Yaskawa INFORM job: kufsa_test_250.JBI

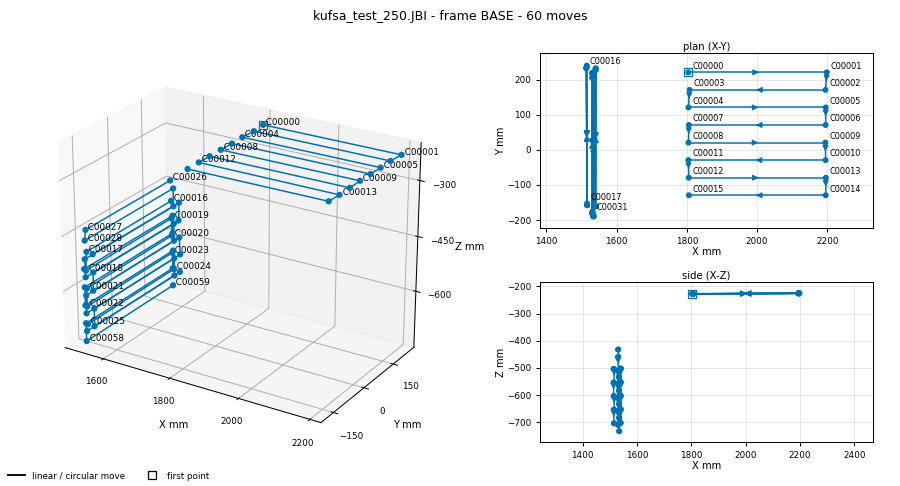
[picture p0: tool path of kufsa_test_250.JBI in frame BASE, 60 of 65 moves have a stored position in this frame; points joined in program order, loops and branches not executed]
/JOB
//NAME kufsa_test_250
//POS
///NPOS 60,0,60,0,0,0
///TOOL 0
///POSTYPE BASE
///RECTAN
///RCONF 0,0,0,0,0,0,0,0,0,0,0,0,0,0,0,0,0,0,0,0,0,0,0,0
C00000=1804.266,220.599,-227.332,179.0000,1.0000,1.0000
C00001=2198.370,220.599,-225.837,179.0000,1.0000,1.0000
C00002=2194.801,170.599,-225.649,179.0000,1.0000,1.0000
C00003=1807.577,170.599,-227.559,179.0000,1.0000,1.0000
C00004=1804.622,120.599,-227.769,179.0000,1.0000,1.0000
C00005=2195.335,120.599,-225.843,179.0000,1.0000,1.0000
C00006=2195.106,70.599,-225.320,179.0000,1.0000,1.0000
C00007=1805.716,70.599,-228.029,179.0000,1.0000,1.0000
C00008=1804.735,20.599,-228.045,179.0000,1.0000,1.0000
C00009=2194.418,20.599,-225.391,179.0000,1.0000,1.0000
C00010=2195.097,-29.400,-225.681,179.0000,1.0000,1.0000
C00011=1804.440,-29.400,-228.141,179.0000,1.0000,1.0000
C00012=1805.619,-79.400,-227.256,179.0000,1.0000,1.0000
C00013=2195.630,-79.400,-225.700,179.0000,1.0000,1.0000
C00014=2195.292,-129.400,-224.241,179.0000,1.0000,1.0000
C00015=1805.953,-129.400,-227.208,179.0000,1.0000,1.0000
C00016=1513.631,232.354,-503.993,179.0000,-89.9999,1.0000
C00017=1516.149,-153.231,-503.993,179.0000,-89.9999,1.0000
C00018=1516.042,-157.471,-553.993,179.0000,-89.9999,1.0000
C00019=1513.923,233.133,-553.993,179.0000,-89.9999,1.0000
C00020=1514.033,233.523,-603.993,179.0000,-89.9999,1.0000
C00021=1516.196,-156.884,-603.993,179.0000,-89.9999,1.0000
C00022=1516.145,-156.999,-653.993,179.0000,-89.9999,1.0000
C00023=1514.649,233.710,-653.993,179.0000,-89.9999,1.0000
C00024=1515.282,239.938,-703.993,179.0000,-89.9999,1.0000
C00025=1516.324,-157.007,-703.993,179.0000,-89.9999,1.0000
C00026=1530.443,204.779,-432.522,179.0000,-89.9999,1.0000
C00027=1531.499,-175.214,-432.522,179.0000,-89.9999,1.0000
C00028=1531.405,-179.918,-459.727,179.0000,-89.9999,1.0000
C00029=1530.485,218.119,-459.727,179.0000,-89.9999,1.0000
C00030=1531.882,216.269,-509.727,179.0000,-89.9999,1.0000
C00031=1531.275,-181.949,-509.727,179.0000,-89.9999,1.0000
C00032=1531.305,-180.389,-559.727,179.0000,-89.9999,1.0000
C00033=1531.688,217.320,-559.727,179.0000,-89.9999,1.0000
C00034=1530.439,218.736,-609.727,179.0000,-89.9999,1.0000
C00035=1531.606,-180.718,-609.727,179.0000,-89.9999,1.0000
C00036=1530.852,-180.562,-659.727,179.0000,-89.9999,1.0000
C00037=1531.645,217.737,-659.727,179.0000,-89.9999,1.0000
C00038=1532.334,216.222,-709.727,179.0000,-89.9999,1.0000
C00039=1530.209,-180.083,-709.727,179.0000,-89.9999,1.0000
C00040=1540.494,-160.372,-502.282,179.0000,-89.9999,1.0000
C00041=1540.352,230.020,-502.282,179.0000,-89.9999,1.0000
C00042=1540.533,226.582,-552.282,179.0000,-89.9999,1.0000
C00043=1540.232,-160.082,-552.282,179.0000,-89.9999,1.0000
C00044=1539.904,-161.733,-602.282,179.0000,-89.9999,1.0000
C00045=1540.218,229.622,-602.282,179.0000,-89.9999,1.0000
C00046=1540.573,232.252,-652.282,179.0000,-89.9999,1.0000
C00047=1540.340,-160.160,-652.282,179.0000,-89.9999,1.0000
C00048=1539.291,-159.918,-702.282,179.0000,-89.9999,1.0000
C00049=1540.509,230.302,-702.282,179.0000,-89.9999,1.0000
C00050=1534.042,-189.208,-533.001,179.0000,-89.9999,1.0000
C00051=1534.110,208.321,-533.001,179.0000,-89.9999,1.0000
C00052=1533.962,207.490,-583.001,179.0000,-89.9999,1.0000
C00053=1534.342,-189.439,-583.001,179.0000,-89.9999,1.0000
C00054=1534.609,-189.394,-633.001,179.0000,-89.9999,1.0000
C00055=1534.722,207.440,-633.001,179.0000,-89.9999,1.0000
C00056=1535.013,204.575,-683.001,179.0000,-89.9999,1.0000
C00057=1534.488,-188.796,-683.001,179.0000,-89.9999,1.0000
C00058=1534.671,-189.015,-733.001,179.0000,-89.9999,1.0000
C00059=1535.183,204.586,-733.001,179.0000,-89.9999,1.0000
///POSTYPE PULSE
///PULSE
EC00000=0
EC00001=0
EC00002=0
EC00003=0
EC00004=0
EC00005=0
EC00006=0
EC00007=0
EC00008=0
EC00009=0
EC00010=0
EC00011=0
EC00012=0
EC00013=0
EC00014=0
EC00015=0
EC00016=0
EC00017=0
EC00018=0
EC00019=0
EC00020=0
EC00021=0
EC00022=0
EC00023=0
EC00024=0
EC00025=0
EC00026=92160
EC00027=92160
EC00028=92160
EC00029=92160
EC00030=92160
EC00031=92160
EC00032=92160
EC00033=92160
EC00034=92160
EC00035=92160
EC00036=92160
EC00037=92160
EC00038=92160
EC00039=92160
EC00040=184320
EC00041=184320
EC00042=184320
EC00043=184320
EC00044=184320
EC00045=184320
EC00046=184320
EC00047=184320
EC00048=184320
EC00049=184320
EC00050=276480
EC00051=276480
EC00052=276480
EC00053=276480
EC00054=276480
EC00055=276480
EC00056=276480
EC00057=276480
EC00058=276480
EC00059=276480
//INST
///DATE 2023/01/18 14:48
///ATTR SC,RW,RJ
////FRAME BASE
///GROUP1 RB1,ST1
NOP
MOVJ C00000 EC00000 VJ=15.00
SPYON
MOVL C00001 EC00001 V=200.0
MOVL C00002 EC00002 V=200.0
MOVL C00003 EC00003 V=200.0
MOVL C00004 EC00004 V=200.0
MOVL C00005 EC00005 V=200.0
MOVL C00006 EC00006 V=200.0
MOVL C00007 EC00007 V=200.0
MOVL C00008 EC00008 V=200.0
MOVL C00009 EC00009 V=200.0
MOVL C00010 EC00010 V=200.0
MOVL C00011 EC00011 V=200.0
MOVL C00012 EC00012 V=200.0
MOVL C00013 EC00013 V=200.0
MOVL C00014 EC00014 V=200.0
MOVL C00015 EC00015 V=200.0
SPYOF
MOVJ P009 VJ=15.00
MOVJ C00016 EC00016 VJ=15.00
SPYON
MOVL C00017 EC00017 V=200.0
MOVL C00018 EC00018 V=200.0
MOVL C00019 EC00019 V=200.0
MOVL C00020 EC00020 V=200.0
MOVL C00021 EC00021 V=200.0
MOVL C00022 EC00022 V=200.0
MOVL C00023 EC00023 V=200.0
MOVL C00024 EC00024 V=200.0
MOVL C00025 EC00025 V=200.0
SPYOF
MOVJ P009 VJ=15.00
MOVJ C00026 EC00026 VJ=15.00
SPYON
MOVL C00027 EC00027 V=200.0
MOVL C00028 EC00028 V=200.0
MOVL C00029 EC00029 V=200.0
MOVL C00030 EC00030 V=200.0
MOVL C00031 EC00031 V=200.0
MOVL C00032 EC00032 V=200.0
MOVL C00033 EC00033 V=200.0
MOVL C00034 EC00034 V=200.0
MOVL C00035 EC00035 V=200.0
MOVL C00036 EC00036 V=200.0
MOVL C00037 EC00037 V=200.0
MOVL C00038 EC00038 V=200.0
MOVL C00039 EC00039 V=200.0
SPYOF
MOVJ P009 VJ=15.00
MOVJ C00040 EC00040 VJ=15.00
SPYON
MOVL C00041 EC00041 V=200.0
MOVL C00042 EC00042 V=200.0
MOVL C00043 EC00043 V=200.0
MOVL C00044 EC00044 V=200.0
MOVL C00045 EC00045 V=200.0
MOVL C00046 EC00046 V=200.0
MOVL C00047 EC00047 V=200.0
MOVL C00048 EC00048 V=200.0
MOVL C00049 EC00049 V=200.0
SPYOF
MOVJ P009 VJ=15.00
MOVJ C00050 EC00050 VJ=15.00
SPYON
MOVL C00051 EC00051 V=200.0
MOVL C00052 EC00052 V=200.0
MOVL C00053 EC00053 V=200.0
MOVL C00054 EC00054 V=200.0
MOVL C00055 EC00055 V=200.0
MOVL C00056 EC00056 V=200.0
MOVL C00057 EC00057 V=200.0
MOVL C00058 EC00058 V=200.0
MOVL C00059 EC00059 V=200.0
SPYOF
MOVJ P009 VJ=15.00
END
